(* CoDeSys 2.3 export: ALARMAND_FB.EXP *)

(* POU FB/ФБ аварий/AlarmAND_FB, ST *)
(* если на обоих входих истина, запускается таймер и по истечении
 указаного времяни присваивает зничение на Out=true на оба выхода.
AlarmAND_FB_Res сбросит Out на false на оба выхода если первое условие and не выполняется*)
FUNCTION_BLOCK AlarmAND_FB
VAR_INPUT
	input: BOOL;
	inversion : BOOL;
END_VAR
VAR_OUTPUT
	bError: BOOL;
END_VAR
VAR
	TON1 : TON;
	SEMA1 : SEMA;
END_VAR
IF NOT  inversion AND input
THEN ton1.IN := TRUE; (*инверсия*)
ELSE  ton1.IN := FALSE;
END_IF

TON1(PT:= T#15s);

SEMA1(
	CLAIM:=ton1.Q ,
	RELEASE:= b0x0); (*if CLAIM=true of SUSY=true, RELEASE reset. Reset возможен только когда   CLAIM=false*)

bError := SEL (sema1.BUSY, FALSE, TRUE);
END_FUNCTION_BLOCK
